PROGRAM Stn051_16_ReturnLnSw
VAR
//should be correct - from TW 
	{attribute 'TcLinkTo' := '.iInfeedSensor := TIIB[N10S08 (EL1008)]^Channel 7^Input;
		.iMachineReady := TIIB[N10S08 (EL1008)]^Channel 8^Input;
		.oBoschInfeedConvFltRst := TIIB[N10S09 (EL2008)]^Channel 4^Output;
		.oIntraloxInfeedConvFltRst := TIIB[N10S09 (EL2008)]^Channel 5^Output;
		.oIntraloxOutfeedConv1FltRst := TIIB[N10S09 (EL2008)]^Channel 6^Output;
		.oIntraloxOutfeedConv2FltRst := TIIB[N10S09 (EL2008)]^Channel 7^Output;
		.oDornerOutfeedConvFltRst := TIIB[N10S09 (EL2008)]^Channel 8^Output;
		.oClearFault := TIIB[N10S10 (EL2008)]^Channel 1^Output;
		.oMotorsRunning := TIIB[N10S10 (EL2008)]^Channel 2^Output;
		.oOutfeedDivertBit[0] := TIIB[N10S10 (EL2008)]^Channel 3^Output;
		.oOutfeedDivertBit[1] := TIIB[N10S10 (EL2008)]^Channel 4^Output;
		.oInfeedBeltBit[0] := TIIB[N10S10 (EL2008)]^Channel 5^Output;
		.oInfeedBeltBit[1] := TIIB[N10S10 (EL2008)]^Channel 6^Output;
		.oBoschInfeedConvRun := TIIB[N10S13 (EL2008)]^Channel 4^Output;
		.oIntraloxInfeedConvRun := TIIB[N10S13 (EL2008)]^Channel 5^Output;
		.oIntraloxOutfeedConv1Run := TIIB[N10S13 (EL2008)]^Channel 6^Output;
		.oIntraloxOutfeedConv2Run := TIIB[N10S13 (EL2008)]^Channel 7^Output;
		.oDornerOutfeedConvRun := TIIB[N10S13 (EL2008)]^Channel 8^Output;
		.iBoschInfeedVFDNotRunning := TIIB[N10S18 (EL1008)]^Channel 1^Input;
		.iBoschInfeedVFDNotFaulted := TIIB[N10S18 (EL1008)]^Channel 2^Input;
		.iIntraloxInfeedVFDNotRunning := TIIB[N10S18 (EL1008)]^Channel 3^Input;
		.iIntraloxInfeedVFDNotFaulted := TIIB[N10S18 (EL1008)]^Channel 4^Input;
		.iIntraloxOutfeedVFD1NotRunning := TIIB[N10S18 (EL1008)]^Channel 5^Input;
		.iIntraloxOutfeedVFD1NotFaulted := TIIB[N10S18 (EL1008)]^Channel 6^Input;
		.iIntraloxOutfeedVFD2NotRunning := TIIB[N10S18 (EL1008)]^Channel 7^Input;
		.iIntraloxOutfeedVFD2NotFaulted := TIIB[N10S18 (EL1008)]^Channel 8^Input;
		.iDornerOutfeedVFDNotRunning := TIIB[N10S19 (EL1008)]^Channel 1^Input;
		.iDornerOutfeedVFDNotFaulted := TIIB[N10S19 (EL1008)]^Channel 2^Input'}
	{attribute 'TcLinkToOSO' := '.iBoschInfeedMtrDiscOK := <0,1,4>TIIB[N13S00 (AL1332)]^N13S01 (AL2341)^TxPDO^input byte 1;
		.iIntraloxInfeedMtrDiscOK := <0,1,4>TIIB[N13S00 (AL1332)]^N13S01 (AL2341)^TxPDO^input byte 3;
		.iIntraloxOutfeedMtr1DiscOK := <0,1,3>TIIB[N13S00 (AL1332)]^N13S03 (AL2341)^TxPDO^input byte 3;
		.iIntraloxOutfeedMtr2DiscOK := <0,1,4>TIIB[N13S00 (AL1332)]^N13S03 (AL2341)^TxPDO^input byte 1;
		.iDornerOutfeedMtrDiscOK := <0,1,4>TIIB[N13S00 (AL1332)]^N13S03 (AL2341)^TxPDO^input byte 3;
		.iBreakStop1PuckPresent[1] := <0,1,0>TIIB[N13S00 (AL1332)]^N13S03 (AL2341)^TxPDO^input byte 0;
		.iBreakStop1PuckPresent[2] := <0,1,2>TIIB[N13S00 (AL1332)]^N13S03 (AL2341)^TxPDO^input byte 0;
		.iBreakStop1PuckPresent[3] := <0,1,4>TIIB[N13S00 (AL1332)]^N13S03 (AL2341)^TxPDO^input byte 0;
		.iBreakStop2PuckPresent[1] := <0,1,1>TIIB[N13S00 (AL1332)]^N13S03 (AL2341)^TxPDO^input byte 0;
		.iBreakStop2PuckPresent[2] := <0,1,3>TIIB[N13S00 (AL1332)]^N13S03 (AL2341)^TxPDO^input byte 0;
		.iBreakStop2PuckPresent[3] := <0,1,0>TIIB[N13S00 (AL1332)]^N13S03 (AL2341)^TxPDO^input byte 1;
		.iBreakStop1BufferFull[1] := <0,1,0>TIIB[N13S00 (AL1332)]^N13S03 (AL2341)^TxPDO^input byte 2;
		.iBreakStop1BufferFull[2] := <0,1,2>TIIB[N13S00 (AL1332)]^N13S03 (AL2341)^TxPDO^input byte 2;
		.iBreakStop1BufferFull[3] := <0,1,4>TIIB[N13S00 (AL1332)]^N13S03 (AL2341)^TxPDO^input byte 2;
		.oBreakStop1PuckRelease[1] := <0,1,4>TIIB[N13S00 (AL1332)]^N13S02 (EX260)^RxPDO^output byte 0;
		.oBreakStop1PuckRelease[2] := <0,1,4>TIIB[N13S00 (AL1332)]^N13S02 (EX260)^RxPDO^output byte 1;
		.oBreakStop1PuckRelease[3] := <0,1,4>TIIB[N13S00 (AL1332)]^N13S02 (EX260)^RxPDO^output byte 2'}
	fb3LaneSwitchMain: FB_3LaneSwitchMain;
	
END_VAR

//  This code instantiates a component that is implimented as a common function block
//    Note that I/O is linked directly to I/O variables inside the named instance

fb3LaneSwitchMain.pWorkStopMain[1] := ADR(gStn051_11_ReturnLnSwPrestopMainGrn);
fb3LaneSwitchMain.pWorkStopMain[2] := ADR(gStn051_13_ReturnLnSwPrestopMainRed);
fb3LaneSwitchMain.pWorkStopMain[3] := ADR(gStn051_15_ReturnLnSwPrestopMainBlu);

fb3LaneSwitchMain(pStn := ADR(gStn051),
	pCmp := ADR(gStn051_16_ReturnLnSw),
	pStateTraceBuffer := ADR(gStn051_StateTraceBuffer),
	pStateTraceFIFO := ADR(gStn051_StateTraceFifo),
	pStats := ADR(gStn051_02_Stats));
	

// Publish Bosch infeed motor running so other station breakstop can decide if ok to release	
gProduced_Stn051ToSafetyInterface.Stn051PLCData[0].10 := gStn051_16_ReturnLnSw.BoschInfeedConvRunning;

END_PROGRAM

(* stored: Version 1.1.0.1, ProductVersion 3.1.4024.6
   POU Stn051_16_ReturnLnSw: Id {1349439e-0158-45a3-80b3-b6c27b015b95}, SpecialFunc None *)
